PROGRAM MAIN
VAR
 fbChangeTime : FB_ChangeSystemTime;
END_VAR

fbChangeTime(systemTime:=GVL_Hmi.systemTime);

END_PROGRAM

(* stored: Version 1.1.0.1, ProductVersion 3.1.4024.3
   POU MAIN: Id {4d4fc665-cc1d-4628-b20d-a2c97b9c8da7}, SpecialFunc None *)
